FUNCTION Convert_LWORD_TO_REAL : Hresult
VAR_INPUT
	in : LWORD;
	out : REFERENCE TO REAL;
END_VAR
VAR
	converted : REAL;
END_VAR
VAR CONSTANT
	INCOMPATIBLE : HRESULT := 16#9811070E;
END_VAR

converted := LWORD_TO_REAL(in);

IF (REAL_TO_LWORD(converted) <> in) THEN
	Convert_LWORD_TO_REAL := INCOMPATIBLE;
	RETURN;
END_IF

out := converted;

END_FUNCTION

(* stored: Version 1.1.0.1, ProductVersion 3.1.4024.12
   POU Convert_LWORD_TO_REAL: Id {b447de2d-addc-4f8d-a746-4482413c51ae}, SpecialFunc None *)
